# EPICS SNL sequencer program: SOFBMonApp/src/SOFBMonOrbit.stt
program SOFBMonOrbit
option +s;

double timeout, window;
int timeout_cnt;

assign timeout to "{P}{R}SlowOrbTimeout-SP";
monitor timeout;
assign window to "{P}{R}SlowOrbWindow-SP";
monitor window;
assign timeout_cnt to "{P}{R}SlowOrbTimeoutCnt-Mon";

float orbit[320];
float orbit_from_bpms[320];

assign orbit to "{P}{R}SlowOrbRaw-Mon";
assign orbit_from_bpms to {
    "SI-01M2:DI-BPM:PosX-Mon",
    "SI-01C1:DI-BPM-1:PosX-Mon",
    "SI-01C1:DI-BPM-2:PosX-Mon",
    "SI-01C2:DI-BPM:PosX-Mon",
    "SI-01C3:DI-BPM-1:PosX-Mon",
    "SI-01C3:DI-BPM-2:PosX-Mon",
    "SI-01C4:DI-BPM:PosX-Mon",
    "SI-02M1:DI-BPM:PosX-Mon",
    "SI-02M2:DI-BPM:PosX-Mon",
    "SI-02C1:DI-BPM-1:PosX-Mon",
    "SI-02C1:DI-BPM-2:PosX-Mon",
    "SI-02C2:DI-BPM:PosX-Mon",
    "SI-02C3:DI-BPM-1:PosX-Mon",
    "SI-02C3:DI-BPM-2:PosX-Mon",
    "SI-02C4:DI-BPM:PosX-Mon",
    "SI-03M1:DI-BPM:PosX-Mon",
    "SI-03M2:DI-BPM:PosX-Mon",
    "SI-03C1:DI-BPM-1:PosX-Mon",
    "SI-03C1:DI-BPM-2:PosX-Mon",
    "SI-03C2:DI-BPM:PosX-Mon",
    "SI-03C3:DI-BPM-1:PosX-Mon",
    "SI-03C3:DI-BPM-2:PosX-Mon",
    "SI-03C4:DI-BPM:PosX-Mon",
    "SI-04M1:DI-BPM:PosX-Mon",
    "SI-04M2:DI-BPM:PosX-Mon",
    "SI-04C1:DI-BPM-1:PosX-Mon",
    "SI-04C1:DI-BPM-2:PosX-Mon",
    "SI-04C2:DI-BPM:PosX-Mon",
    "SI-04C3:DI-BPM-1:PosX-Mon",
    "SI-04C3:DI-BPM-2:PosX-Mon",
    "SI-04C4:DI-BPM:PosX-Mon",
    "SI-05M1:DI-BPM:PosX-Mon",
    "SI-05M2:DI-BPM:PosX-Mon",
    "SI-05C1:DI-BPM-1:PosX-Mon",
    "SI-05C1:DI-BPM-2:PosX-Mon",
    "SI-05C2:DI-BPM:PosX-Mon",
    "SI-05C3:DI-BPM-1:PosX-Mon",
    "SI-05C3:DI-BPM-2:PosX-Mon",
    "SI-05C4:DI-BPM:PosX-Mon",
    "SI-06M1:DI-BPM:PosX-Mon",
    "SI-06M2:DI-BPM:PosX-Mon",
    "SI-06C1:DI-BPM-1:PosX-Mon",
    "SI-06C1:DI-BPM-2:PosX-Mon",
    "SI-06C2:DI-BPM:PosX-Mon",
    "SI-06C3:DI-BPM-1:PosX-Mon",
    "SI-06C3:DI-BPM-2:PosX-Mon",
    "SI-06C4:DI-BPM:PosX-Mon",
    "SI-07M1:DI-BPM:PosX-Mon",
    "SI-07M2:DI-BPM:PosX-Mon",
    "SI-07C1:DI-BPM-1:PosX-Mon",
    "SI-07C1:DI-BPM-2:PosX-Mon",
    "SI-07C2:DI-BPM:PosX-Mon",
    "SI-07C3:DI-BPM-1:PosX-Mon",
    "SI-07C3:DI-BPM-2:PosX-Mon",
    "SI-07C4:DI-BPM:PosX-Mon",
    "SI-08M1:DI-BPM:PosX-Mon",
    "SI-08M2:DI-BPM:PosX-Mon",
    "SI-08C1:DI-BPM-1:PosX-Mon",
    "SI-08C1:DI-BPM-2:PosX-Mon",
    "SI-08C2:DI-BPM:PosX-Mon",
    "SI-08C3:DI-BPM-1:PosX-Mon",
    "SI-08C3:DI-BPM-2:PosX-Mon",
    "SI-08C4:DI-BPM:PosX-Mon",
    "SI-09M1:DI-BPM:PosX-Mon",
    "SI-09M2:DI-BPM:PosX-Mon",
    "SI-09C1:DI-BPM-1:PosX-Mon",
    "SI-09C1:DI-BPM-2:PosX-Mon",
    "SI-09C2:DI-BPM:PosX-Mon",
    "SI-09C3:DI-BPM-1:PosX-Mon",
    "SI-09C3:DI-BPM-2:PosX-Mon",
    "SI-09C4:DI-BPM:PosX-Mon",
    "SI-10M1:DI-BPM:PosX-Mon",
    "SI-10M2:DI-BPM:PosX-Mon",
    "SI-10C1:DI-BPM-1:PosX-Mon",
    "SI-10C1:DI-BPM-2:PosX-Mon",
    "SI-10C2:DI-BPM:PosX-Mon",
    "SI-10C3:DI-BPM-1:PosX-Mon",
    "SI-10C3:DI-BPM-2:PosX-Mon",
    "SI-10C4:DI-BPM:PosX-Mon",
    "SI-11M1:DI-BPM:PosX-Mon",
    "SI-11M2:DI-BPM:PosX-Mon",
    "SI-11C1:DI-BPM-1:PosX-Mon",
    "SI-11C1:DI-BPM-2:PosX-Mon",
    "SI-11C2:DI-BPM:PosX-Mon",
    "SI-11C3:DI-BPM-1:PosX-Mon",
    "SI-11C3:DI-BPM-2:PosX-Mon",
    "SI-11C4:DI-BPM:PosX-Mon",
    "SI-12M1:DI-BPM:PosX-Mon",
    "SI-12M2:DI-BPM:PosX-Mon",
    "SI-12C1:DI-BPM-1:PosX-Mon",
    "SI-12C1:DI-BPM-2:PosX-Mon",
    "SI-12C2:DI-BPM:PosX-Mon",
    "SI-12C3:DI-BPM-1:PosX-Mon",
    "SI-12C3:DI-BPM-2:PosX-Mon",
    "SI-12C4:DI-BPM:PosX-Mon",
    "SI-13M1:DI-BPM:PosX-Mon",
    "SI-13M2:DI-BPM:PosX-Mon",
    "SI-13C1:DI-BPM-1:PosX-Mon",
    "SI-13C1:DI-BPM-2:PosX-Mon",
    "SI-13C2:DI-BPM:PosX-Mon",
    "SI-13C3:DI-BPM-1:PosX-Mon",
    "SI-13C3:DI-BPM-2:PosX-Mon",
    "SI-13C4:DI-BPM:PosX-Mon",
    "SI-14M1:DI-BPM:PosX-Mon",
    "SI-14M2:DI-BPM:PosX-Mon",
    "SI-14C1:DI-BPM-1:PosX-Mon",
    "SI-14C1:DI-BPM-2:PosX-Mon",
    "SI-14C2:DI-BPM:PosX-Mon",
    "SI-14C3:DI-BPM-1:PosX-Mon",
    "SI-14C3:DI-BPM-2:PosX-Mon",
    "SI-14C4:DI-BPM:PosX-Mon",
    "SI-15M1:DI-BPM:PosX-Mon",
    "SI-15M2:DI-BPM:PosX-Mon",
    "SI-15C1:DI-BPM-1:PosX-Mon",
    "SI-15C1:DI-BPM-2:PosX-Mon",
    "SI-15C2:DI-BPM:PosX-Mon",
    "SI-15C3:DI-BPM-1:PosX-Mon",
    "SI-15C3:DI-BPM-2:PosX-Mon",
    "SI-15C4:DI-BPM:PosX-Mon",
    "SI-16M1:DI-BPM:PosX-Mon",
    "SI-16M2:DI-BPM:PosX-Mon",
    "SI-16C1:DI-BPM-1:PosX-Mon",
    "SI-16C1:DI-BPM-2:PosX-Mon",
    "SI-16C2:DI-BPM:PosX-Mon",
    "SI-16C3:DI-BPM-1:PosX-Mon",
    "SI-16C3:DI-BPM-2:PosX-Mon",
    "SI-16C4:DI-BPM:PosX-Mon",
    "SI-17M1:DI-BPM:PosX-Mon",
    "SI-17M2:DI-BPM:PosX-Mon",
    "SI-17C1:DI-BPM-1:PosX-Mon",
    "SI-17C1:DI-BPM-2:PosX-Mon",
    "SI-17C2:DI-BPM:PosX-Mon",
    "SI-17C3:DI-BPM-1:PosX-Mon",
    "SI-17C3:DI-BPM-2:PosX-Mon",
    "SI-17C4:DI-BPM:PosX-Mon",
    "SI-18M1:DI-BPM:PosX-Mon",
    "SI-18M2:DI-BPM:PosX-Mon",
    "SI-18C1:DI-BPM-1:PosX-Mon",
    "SI-18C1:DI-BPM-2:PosX-Mon",
    "SI-18C2:DI-BPM:PosX-Mon",
    "SI-18C3:DI-BPM-1:PosX-Mon",
    "SI-18C3:DI-BPM-2:PosX-Mon",
    "SI-18C4:DI-BPM:PosX-Mon",
    "SI-19M1:DI-BPM:PosX-Mon",
    "SI-19M2:DI-BPM:PosX-Mon",
    "SI-19C1:DI-BPM-1:PosX-Mon",
    "SI-19C1:DI-BPM-2:PosX-Mon",
    "SI-19C2:DI-BPM:PosX-Mon",
    "SI-19C3:DI-BPM-1:PosX-Mon",
    "SI-19C3:DI-BPM-2:PosX-Mon",
    "SI-19C4:DI-BPM:PosX-Mon",
    "SI-20M1:DI-BPM:PosX-Mon",
    "SI-20M2:DI-BPM:PosX-Mon",
    "SI-20C1:DI-BPM-1:PosX-Mon",
    "SI-20C1:DI-BPM-2:PosX-Mon",
    "SI-20C2:DI-BPM:PosX-Mon",
    "SI-20C3:DI-BPM-1:PosX-Mon",
    "SI-20C3:DI-BPM-2:PosX-Mon",
    "SI-20C4:DI-BPM:PosX-Mon",
    "SI-01M1:DI-BPM:PosX-Mon",
    "SI-01M2:DI-BPM:PosY-Mon",
    "SI-01C1:DI-BPM-1:PosY-Mon",
    "SI-01C1:DI-BPM-2:PosY-Mon",
    "SI-01C2:DI-BPM:PosY-Mon",
    "SI-01C3:DI-BPM-1:PosY-Mon",
    "SI-01C3:DI-BPM-2:PosY-Mon",
    "SI-01C4:DI-BPM:PosY-Mon",
    "SI-02M1:DI-BPM:PosY-Mon",
    "SI-02M2:DI-BPM:PosY-Mon",
    "SI-02C1:DI-BPM-1:PosY-Mon",
    "SI-02C1:DI-BPM-2:PosY-Mon",
    "SI-02C2:DI-BPM:PosY-Mon",
    "SI-02C3:DI-BPM-1:PosY-Mon",
    "SI-02C3:DI-BPM-2:PosY-Mon",
    "SI-02C4:DI-BPM:PosY-Mon",
    "SI-03M1:DI-BPM:PosY-Mon",
    "SI-03M2:DI-BPM:PosY-Mon",
    "SI-03C1:DI-BPM-1:PosY-Mon",
    "SI-03C1:DI-BPM-2:PosY-Mon",
    "SI-03C2:DI-BPM:PosY-Mon",
    "SI-03C3:DI-BPM-1:PosY-Mon",
    "SI-03C3:DI-BPM-2:PosY-Mon",
    "SI-03C4:DI-BPM:PosY-Mon",
    "SI-04M1:DI-BPM:PosY-Mon",
    "SI-04M2:DI-BPM:PosY-Mon",
    "SI-04C1:DI-BPM-1:PosY-Mon",
    "SI-04C1:DI-BPM-2:PosY-Mon",
    "SI-04C2:DI-BPM:PosY-Mon",
    "SI-04C3:DI-BPM-1:PosY-Mon",
    "SI-04C3:DI-BPM-2:PosY-Mon",
    "SI-04C4:DI-BPM:PosY-Mon",
    "SI-05M1:DI-BPM:PosY-Mon",
    "SI-05M2:DI-BPM:PosY-Mon",
    "SI-05C1:DI-BPM-1:PosY-Mon",
    "SI-05C1:DI-BPM-2:PosY-Mon",
    "SI-05C2:DI-BPM:PosY-Mon",
    "SI-05C3:DI-BPM-1:PosY-Mon",
    "SI-05C3:DI-BPM-2:PosY-Mon",
    "SI-05C4:DI-BPM:PosY-Mon",
    "SI-06M1:DI-BPM:PosY-Mon",
    "SI-06M2:DI-BPM:PosY-Mon",
    "SI-06C1:DI-BPM-1:PosY-Mon",
    "SI-06C1:DI-BPM-2:PosY-Mon",
    "SI-06C2:DI-BPM:PosY-Mon",
    "SI-06C3:DI-BPM-1:PosY-Mon",
    "SI-06C3:DI-BPM-2:PosY-Mon",
    "SI-06C4:DI-BPM:PosY-Mon",
    "SI-07M1:DI-BPM:PosY-Mon",
    "SI-07M2:DI-BPM:PosY-Mon",
    "SI-07C1:DI-BPM-1:PosY-Mon",
    "SI-07C1:DI-BPM-2:PosY-Mon",
    "SI-07C2:DI-BPM:PosY-Mon",
    "SI-07C3:DI-BPM-1:PosY-Mon",
    "SI-07C3:DI-BPM-2:PosY-Mon",
    "SI-07C4:DI-BPM:PosY-Mon",
    "SI-08M1:DI-BPM:PosY-Mon",
    "SI-08M2:DI-BPM:PosY-Mon",
    "SI-08C1:DI-BPM-1:PosY-Mon",
    "SI-08C1:DI-BPM-2:PosY-Mon",
    "SI-08C2:DI-BPM:PosY-Mon",
    "SI-08C3:DI-BPM-1:PosY-Mon",
    "SI-08C3:DI-BPM-2:PosY-Mon",
    "SI-08C4:DI-BPM:PosY-Mon",
    "SI-09M1:DI-BPM:PosY-Mon",
    "SI-09M2:DI-BPM:PosY-Mon",
    "SI-09C1:DI-BPM-1:PosY-Mon",
    "SI-09C1:DI-BPM-2:PosY-Mon",
    "SI-09C2:DI-BPM:PosY-Mon",
    "SI-09C3:DI-BPM-1:PosY-Mon",
    "SI-09C3:DI-BPM-2:PosY-Mon",
    "SI-09C4:DI-BPM:PosY-Mon",
    "SI-10M1:DI-BPM:PosY-Mon",
    "SI-10M2:DI-BPM:PosY-Mon",
    "SI-10C1:DI-BPM-1:PosY-Mon",
    "SI-10C1:DI-BPM-2:PosY-Mon",
    "SI-10C2:DI-BPM:PosY-Mon",
    "SI-10C3:DI-BPM-1:PosY-Mon",
    "SI-10C3:DI-BPM-2:PosY-Mon",
    "SI-10C4:DI-BPM:PosY-Mon",
    "SI-11M1:DI-BPM:PosY-Mon",
    "SI-11M2:DI-BPM:PosY-Mon",
    "SI-11C1:DI-BPM-1:PosY-Mon",
    "SI-11C1:DI-BPM-2:PosY-Mon",
    "SI-11C2:DI-BPM:PosY-Mon",
    "SI-11C3:DI-BPM-1:PosY-Mon",
    "SI-11C3:DI-BPM-2:PosY-Mon",
    "SI-11C4:DI-BPM:PosY-Mon",
    "SI-12M1:DI-BPM:PosY-Mon",
    "SI-12M2:DI-BPM:PosY-Mon",
    "SI-12C1:DI-BPM-1:PosY-Mon",
    "SI-12C1:DI-BPM-2:PosY-Mon",
    "SI-12C2:DI-BPM:PosY-Mon",
    "SI-12C3:DI-BPM-1:PosY-Mon",
    "SI-12C3:DI-BPM-2:PosY-Mon",
    "SI-12C4:DI-BPM:PosY-Mon",
    "SI-13M1:DI-BPM:PosY-Mon",
    "SI-13M2:DI-BPM:PosY-Mon",
    "SI-13C1:DI-BPM-1:PosY-Mon",
    "SI-13C1:DI-BPM-2:PosY-Mon",
    "SI-13C2:DI-BPM:PosY-Mon",
    "SI-13C3:DI-BPM-1:PosY-Mon",
    "SI-13C3:DI-BPM-2:PosY-Mon",
    "SI-13C4:DI-BPM:PosY-Mon",
    "SI-14M1:DI-BPM:PosY-Mon",
    "SI-14M2:DI-BPM:PosY-Mon",
    "SI-14C1:DI-BPM-1:PosY-Mon",
    "SI-14C1:DI-BPM-2:PosY-Mon",
    "SI-14C2:DI-BPM:PosY-Mon",
    "SI-14C3:DI-BPM-1:PosY-Mon",
    "SI-14C3:DI-BPM-2:PosY-Mon",
    "SI-14C4:DI-BPM:PosY-Mon",
    "SI-15M1:DI-BPM:PosY-Mon",
    "SI-15M2:DI-BPM:PosY-Mon",
    "SI-15C1:DI-BPM-1:PosY-Mon",
    "SI-15C1:DI-BPM-2:PosY-Mon",
    "SI-15C2:DI-BPM:PosY-Mon",
    "SI-15C3:DI-BPM-1:PosY-Mon",
    "SI-15C3:DI-BPM-2:PosY-Mon",
    "SI-15C4:DI-BPM:PosY-Mon",
    "SI-16M1:DI-BPM:PosY-Mon",
    "SI-16M2:DI-BPM:PosY-Mon",
    "SI-16C1:DI-BPM-1:PosY-Mon",
    "SI-16C1:DI-BPM-2:PosY-Mon",
    "SI-16C2:DI-BPM:PosY-Mon",
    "SI-16C3:DI-BPM-1:PosY-Mon",
    "SI-16C3:DI-BPM-2:PosY-Mon",
    "SI-16C4:DI-BPM:PosY-Mon",
    "SI-17M1:DI-BPM:PosY-Mon",
    "SI-17M2:DI-BPM:PosY-Mon",
    "SI-17C1:DI-BPM-1:PosY-Mon",
    "SI-17C1:DI-BPM-2:PosY-Mon",
    "SI-17C2:DI-BPM:PosY-Mon",
    "SI-17C3:DI-BPM-1:PosY-Mon",
    "SI-17C3:DI-BPM-2:PosY-Mon",
    "SI-17C4:DI-BPM:PosY-Mon",
    "SI-18M1:DI-BPM:PosY-Mon",
    "SI-18M2:DI-BPM:PosY-Mon",
    "SI-18C1:DI-BPM-1:PosY-Mon",
    "SI-18C1:DI-BPM-2:PosY-Mon",
    "SI-18C2:DI-BPM:PosY-Mon",
    "SI-18C3:DI-BPM-1:PosY-Mon",
    "SI-18C3:DI-BPM-2:PosY-Mon",
    "SI-18C4:DI-BPM:PosY-Mon",
    "SI-19M1:DI-BPM:PosY-Mon",
    "SI-19M2:DI-BPM:PosY-Mon",
    "SI-19C1:DI-BPM-1:PosY-Mon",
    "SI-19C1:DI-BPM-2:PosY-Mon",
    "SI-19C2:DI-BPM:PosY-Mon",
    "SI-19C3:DI-BPM-1:PosY-Mon",
    "SI-19C3:DI-BPM-2:PosY-Mon",
    "SI-19C4:DI-BPM:PosY-Mon",
    "SI-20M1:DI-BPM:PosY-Mon",
    "SI-20M2:DI-BPM:PosY-Mon",
    "SI-20C1:DI-BPM-1:PosY-Mon",
    "SI-20C1:DI-BPM-2:PosY-Mon",
    "SI-20C2:DI-BPM:PosY-Mon",
    "SI-20C3:DI-BPM-1:PosY-Mon",
    "SI-20C3:DI-BPM-2:PosY-Mon",
    "SI-20C4:DI-BPM:PosY-Mon",
    "SI-01M1:DI-BPM:PosY-Mon"
};
monitor orbit_from_bpms;

evflag orbit_from_bpms_event;
sync orbit_from_bpms to orbit_from_bpms_event;

%%#include <math.h>
%%#include <stdio.h>

%%#include <epicsTime.h>

entry {
    pvPut(timeout_cnt, ASYNC);
}

ss scan {

    struct epicsTimeStamp sentinels[320] = {0};

    state wait {
        int go_to_read_all;
        entry {
            go_to_read_all = 0;
        }

        when (go_to_read_all) {
        } state read_all

        when (efTest(orbit_from_bpms_event)) {
            struct epicsTimeStamp ts[320];
            int i;
            for (i = 0; i < 320; i++) {
                ts[i] = pvTimeStamp(orbit_from_bpms[i]);
                if (epicsTimeGreaterThan(ts+i, sentinels+i)) {
                    go_to_read_all = 1;
                    break;
                }
            }
        } state wait
    }

    state read_all {
        option -t; /* make delays inside the same state work */

        double spread;
        entry {
            spread = INFINITY;
        }

        when (delay(timeout)) {
            if (pvPutComplete(orbit)) pvPut(orbit, ASYNC);

            timeout_cnt++;
            if (pvPutComplete(timeout_cnt)) pvPut(timeout_cnt, ASYNC);
        } state wait

        when (spread <= window) {
            if (pvPutComplete(orbit)) pvPut(orbit, ASYNC);
        } state wait

        when (efTestAndClear(orbit_from_bpms_event)) {
            struct epicsTimeStamp ts[320];
            int max_idx = 0, min_idx = 0, i;
            for (i = 0; i < 320; i++) {
                ts[i] = pvTimeStamp(orbit_from_bpms[i]);
                if (i > 0) {
                    if (epicsTimeLessThan(ts+i, ts+min_idx)) min_idx = i;
                    else if (epicsTimeGreaterThan(ts+i, ts+max_idx)) max_idx = i;
                }

                /* get orbit ready for pvPut here, since PV monitors can be posted between transitions */
                if (epicsTimeGreaterThan(ts+i, sentinels+i)) {
                    sentinels[i] = ts[i];
                    orbit[i] = orbit_from_bpms[i] / 1000; /* convert to um */
                }
            }
            spread = epicsTimeDiffInSeconds(ts+max_idx, ts+min_idx);
        } state read_all
    }

}
